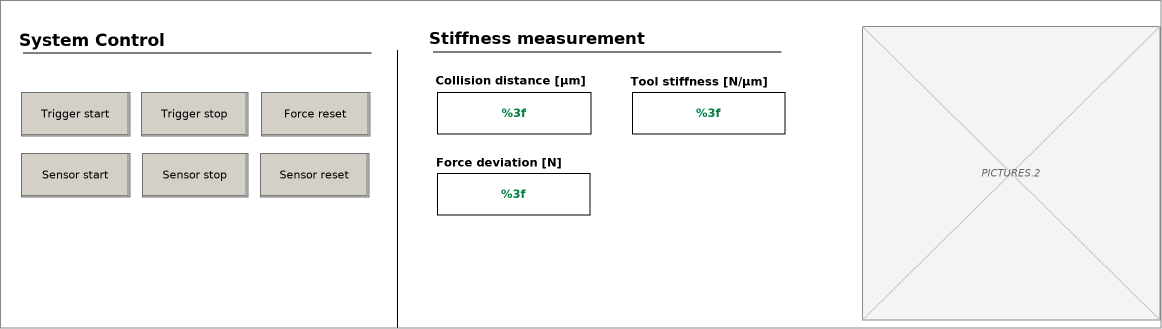
VISUALIZATION VISUALISATION_STIFFNESS_COLLISION  // 1162x329
    Button (21,92 109x44), "Trigger start"
        OnMouseClick: execute { VARIABLES.CAN_TRIGGER_STATE:=1; }
    Button (141,92 107x44), "Trigger stop"
        OnMouseClick: execute { VARIABLES.CAN_TRIGGER_STATE:=0; }
    Button (21,153 109x44), "Sensor start"
        OnMouseClick: execute { CAN_CONTROL_STATE:=1; }
    Button (142,153 106x44), "Sensor stop"
        OnMouseClick: execute { CAN_CONTROL_STATE:=0; }
    Button (260,153 109x44), "Sensor reset"
        OnMouseClick: execute { CAN_CONTROL_STATE:=2; }
    Button (261,92 109x44), "Force reset"
        OnMouseClick: execute { VARIABLES.FORCE_RESET:=1; }
    Rectangle (17,25 150x30), "System Control"
    Line (371,53) (23,53)
    Rectangle (428,31 218x15), "Stiffness measurement"
    Rectangle (632,92 153x42), "%3f", text variable: VARIABLES.TOOL_STIFFNESS_SELC_PTS[1,3]
    Rectangle (437,92 154x42), "%3f", text variable: VARIABLES.COLLISION_DISTANCE
    Rectangle (437,173 153x42), "%3f", text variable: VARIABLES.FORCE_DEVIATION[1]
    Rectangle (437,73 148x15), "Collision distance [µm]"
    Rectangle (437,155 124x15), "Force deviation [N]"
    Rectangle (632,74 135x15), "Tool stiffness [N/µm]"
    Line (397,50) (397,327)
    Line (781,52) (433,52)
    Image (862,26 298x294), image: PICTURES.2
END_VISUALIZATION

(* stored: Version 1.1.0.1, ProductVersion 3.1.0.26
   Visu VISUALISATION_STIFFNESS_COLLISION: Id {24ec0232-0eba-4857-a4de-4d8d1a928b43} *)
